TYPE ST_Camera_CMD :
STRUCT
	
	Inspect1			: BOOL;		
	Inspect2			: BOOL;		
	
END_STRUCT
END_TYPE

(* stored: Version 1.1.0.1, ProductVersion 3.1.4026.17
   DUT ST_Camera_CMD: Id {b04f1e4d-e0a9-4657-bf3c-f43eae8c4118} *)
